ABB RAPID module: Module1.mod

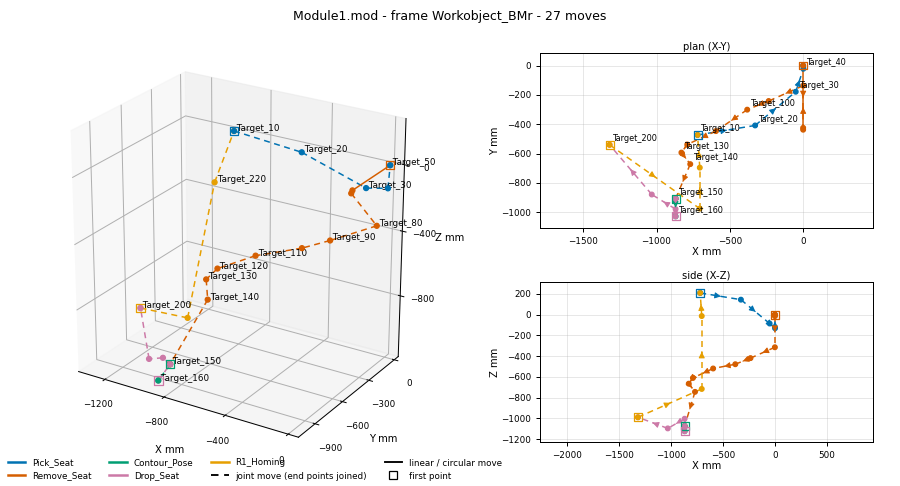
[picture p0: tool path of Module1.mod in frame Workobject_BMr, 27 of 27 moves have a stored position in this frame; points joined in program order, loops and branches not executed]
MODULE Module1
        CONST robtarget Target_10:=[[-720.000011645,-473.523933138,210.010702888],[0.92387952,-0.382683462,-0.000000001,-0.000000014],[0,0,-2,0],[9E+09,9E+09,9E+09,9E+09,9E+09,9E+09]];
    CONST robtarget Target_20:=[[-327.539401228,-408.673770013,145.160539627],[0.923879533,-0.38268343,0.000000079,0.000000068],[0,0,-2,0],[9E+09,9E+09,9E+09,9E+09,9E+09,9E+09]];
    CONST robtarget Target_30:=[[-50.570211496,-178.729757776,-84.783473092],[0.923879521,-0.38268346,0.000000078,0.000000082],[0,0,-2,0],[9E+09,9E+09,9E+09,9E+09,9E+09,9E+09]];
    CONST robtarget Target_40:=[[1.630688405,-21.601801336,-129.840396081],[0.986021938,-0.16291226,0.034630621,0.00458843],[0,1,-3,0],[9E+09,9E+09,9E+09,9E+09,9E+09,9E+09]];
    CONST robtarget Target_50:=[[0,0,0],[1,0,0,0],[0,1,-3,0],[9E+09,9E+09,9E+09,9E+09,9E+09,9E+09]];
    CONST robtarget Target_60:=[[-0.000015252,-424.973966342,-0.707148714],[1,0.000000044,0,-0.000000007],[-1,1,-2,0],[9E+09,9E+09,9E+09,9E+09,9E+09,9E+09]];
    CONST robtarget Target_70:=[[-0.00002672,-437.725095103,-13.4582561],[0.932323884,0.361624356,0.000000045,-0.000000054],[0,1,-3,0],[9E+09,9E+09,9E+09,9E+09,9E+09,9E+09]];
    CONST robtarget Target_80:=[[-0.000202289,-137.474362073,-313.70898176],[0.932323889,0.361624344,0.000000031,-0.000000102],[0,1,-3,0],[9E+09,9E+09,9E+09,9E+09,9E+09,9E+09]];
    CONST robtarget Target_90:=[[-235.078418184,-242.081109941,-418.315728751],[0.909612824,0.35281531,0.088528201,-0.200720267],[-1,1,-3,0],[9E+09,9E+09,9E+09,9E+09,9E+09,9E+09]];
    CONST robtarget Target_100:=[[-381.50057449,-301.005304242,-477.23998966],[0.785975234,0.304859992,0.217055083,-0.492128447],[-1,1,-3,0],[9E+09,9E+09,9E+09,9E+09,9E+09,9E+09]];
    CONST robtarget Target_110:=[[-595.204590481,-447.29356816,-518.353757909],[0.356701612,0.138355938,0.372842374,-0.845346177],[-1,1,-3,0],[9E+09,9E+09,9E+09,9E+09,9E+09,9E+09]];
    CONST robtarget Target_120:=[[-790.24176618,-538.516731861,-609.577038128],[0.181502567,0.070400839,0.395824537,-0.897453885],[-1,1,-3,0],[9E+09,9E+09,9E+09,9E+09,9E+09,9E+09]];
    CONST robtarget Target_130:=[[-830.241673059,-593.670942501,-664.730708999],[0.614428896,0.238321627,0.303513559,-0.688156562],[-1,1,-3,0],[9E+09,9E+09,9E+09,9E+09,9E+09,9E+09]];
    CONST robtarget Target_140:=[[-769.999985431,-672.517919064,-743.579309517],[0.932323793,0.361624592,0.000000012,0.000000047],[-1,1,-2,0],[9E+09,9E+09,9E+09,9E+09,9E+09,9E+09]];
    CONST robtarget Target_150:=[[-870.000060072,-908.394559899,-1073.388035751],[0.923879541,0.382683412,-0.00000002,-0.000000064],[-2,2,-2,0],[9E+09,9E+09,9E+09,9E+09,9E+09,9E+09]];
    CONST robtarget Target_160:=[[-870.000071699,-1028.602739301,-1122.885548688],[0.000000021,-0.000000046,-0.707106773,0.70710679],[-2,2,-4,0],[9E+09,9E+09,9E+09,9E+09,9E+09,9E+09]];
    CONST robtarget Target_170:=[[-870.000060072,-908.394559899,-1073.388035751],[0.923879541,0.382683412,-0.00000002,-0.000000064],[-2,2,-2,0],[9E+09,9E+09,9E+09,9E+09,9E+09,9E+09]];
    CONST robtarget Target_180:=[[-870.000060314,-979.105267008,-1002.677339202],[0.923879518,0.382683467,-0.000000023,-0.000000058],[-2,2,-2,0],[9E+09,9E+09,9E+09,9E+09,9E+09,9E+09]];
    CONST robtarget Target_190:=[[-1032.407360447,-879.660575119,-1095.853940976],[0.70773277,0.293152543,-0.585543817,-0.265168534],[-2,-2,-2,0],[9E+09,9E+09,9E+09,9E+09,9E+09,9E+09]];
    CONST robtarget Target_200:=[[-1319.999841618,-540.699095016,-988.535255888],[0.326505535,0.627211262,-0.212631127,-0.674379843],[-2,-2,-2,0],[9E+09,9E+09,9E+09,9E+09,9E+09,9E+09]];
    CONST robtarget Target_210:=[[-705,-975.712504043,-715.610231087],[0.707047756,0.009131454,0.707047878,0.009131526],[-2,0,-2,0],[9E+09,9E+09,9E+09,9E+09,9E+09,9E+09]];
    CONST robtarget Target_220:=[[-705,-696.262640401,-12.727892234],[0.653281412,-0.270598059,0.653281553,-0.270598041],[-1,0,-2,0],[9E+09,9E+09,9E+09,9E+09,9E+09,9E+09]];
!***********************************************************
    !
    ! Módulo:  Module1
    !
    ! Descripción:
    !   <Introduzca la descripción aquí>
    !
    ! Autor: David
    !
    ! Versión: 1.0
    !
    !***********************************************************


    !***********************************************************
    !
    ! Procedimiento Main
    !
    !   Este es el punto de entrada de su programa
    !
    !***********************************************************
    PROC main()
        Beginning:
        PulseDO Start;
        WaitDI R1_Start,1;
        Pick_Seat;
        WaitTime 2;
        PulseDO R1_Remove;
        Remove_Seat;
        PulseDO Cut_Holes;
        WaitDI To_Contour_Pose,1;
        Contour_Pose;
        PulseDO Cut_Contours;
        WaitDI To_Drop_Pose,1;
        Drop_Seat;
        WaitTime 1;
        PulseDO R1_Drop;
        WaitTime 1;
        R1_Homing;
        GOTO Beginning;
    ENDPROC
    PROC Pick_Seat()
        MoveJ Target_10,v400,z5,tGripper\WObj:=Workobject_BMr;
        MoveJ Target_20,v400,z5,tGripper\WObj:=Workobject_BMr;
        MoveJ Target_30,v400,z5,tGripper\WObj:=Workobject_BMr;
        MoveJ Target_40,v400,z5,tGripper\WObj:=Workobject_BMr;
        MoveJ Target_50,v400,fine,tGripper\WObj:=Workobject_BMr;
    ENDPROC
    PROC Remove_Seat()
        MoveJ Target_50,v400,fine,tGripper\WObj:=Workobject_BMr;
        MoveL Target_60,v300,z5,tGripper\WObj:=Workobject_BMr;
        MoveJ Target_70,v400,z5,tGripper\WObj:=Workobject_BMr;
        MoveJ Target_80,v400,z5,tGripper\WObj:=Workobject_BMr;
        MoveJ Target_90,v400,z5,tGripper\WObj:=Workobject_BMr;
        MoveJ Target_100,v400,z5,tGripper\WObj:=Workobject_BMr;
        MoveJ Target_110,v400,z5,tGripper\WObj:=Workobject_BMr;
        MoveJ Target_120,v400,z5,tGripper\WObj:=Workobject_BMr;
        MoveJ Target_130,v400,z5,tGripper\WObj:=Workobject_BMr;
        MoveJ Target_140,v400,z5,tGripper\WObj:=Workobject_BMr;
        MoveJ Target_150,v400,fine,tGripper\WObj:=Workobject_BMr;
    ENDPROC
    PROC Contour_Pose()
        MoveJ Target_150,v400,fine,tGripper\WObj:=Workobject_BMr;
        MoveJ Target_160,v400,fine,tGripper\WObj:=Workobject_BMr;
    ENDPROC
    PROC Drop_Seat()
        MoveJ Target_160,v1500,z5,tGripper\WObj:=Workobject_BMr;
        MoveJ Target_170,v1500,z5,tGripper\WObj:=Workobject_BMr;
        MoveJ Target_180,v1500,z5,tGripper\WObj:=Workobject_BMr;
        MoveJ Target_190,v1500,z5,tGripper\WObj:=Workobject_BMr;
        MoveJ Target_200,v1500,z5,tGripper\WObj:=Workobject_BMr;
    ENDPROC
    PROC R1_Homing()
        MoveJ Target_200,v400,z5,tGripper\WObj:=Workobject_BMr;
        MoveJ Target_210,v400,z10,tGripper\WObj:=Workobject_BMr;
        MoveJ Target_220,v400,z10,tGripper\WObj:=Workobject_BMr;
        MoveJ Target_10,v400,fine,tGripper\WObj:=Workobject_BMr;
    ENDPROC
ENDMODULE
